FUNCTION_BLOCK FB_IdPool
VAR_INPUT
END_VAR
VAR_OUTPUT
END_VAR
VAR
	aNodes : ARRAY[1..cMaxObjects] OF ST_IdNode;
	pHead : POINTER TO ST_IdNode;
	pTail : POINTER TO ST_IdNode;
END_VAR

METHOD M_GetId : UINT
VAR_INPUT
END_VAR

VAR
	pNode : POINTER TO ST_IdNode;
END_VAR
IF pHead > 0 THEN
	pNode := pHead;
	M_GetId := pNode^.nId;
	IF pHead = pTail THEN //die letzte freie Id
		pHead := 0;
		pTail := 0;
	ELSE
		pHead := pNode^.pNext;
	END_IF
	memset(pNode,0,SIZEOF(ST_IdNode));
END_IF
END_METHOD

METHOD M_ReleaseId : BOOL
VAR_INPUT
	nId : UINT;
END_VAR
//Id in Benutzung?
IF nId >= 0 AND nId <= cMaxObjects AND_THEN aNodes[nId].nId = 0 THEN
	aNodes[nId].nId := nId;
	aNodes[nId].pNext := pHead;
	pHead := ADR(aNodes[nId]);
	M_ReleaseId := TRUE;
END_IF
END_METHOD

METHOD M_Reset : BOOL
VAR_INPUT
END_VAR

VAR
	i : UINT;
END_VAR
pHead := ADR(aNodes[1]);
pTail := ADR(aNodes[cMaxObjects]);
FOR i := 1 TO cMaxObjects BY 1 DO
	aNodes[i].nId := i;
	IF i < cMaxObjects THEN
		aNodes[i].pNext := ADR(aNodes[i+1]);
	ELSE
		aNodes[i].pNext := 0;
	END_IF
END_FOR
END_METHOD

END_FUNCTION_BLOCK

(* stored: Version 1.1.0.1, ProductVersion 3.1.4022.12
   POU FB_IdPool: Id {9849b2e5-dcee-4ced-81f0-c68734dbe188}, SpecialFunc None
   Method M_GetId: Id {e65a9dbd-6f70-4b71-8983-d548273ccf2e}
   Method M_ReleaseId: Id {99864b0b-dddb-4bbb-beb9-6636cb494557}
   Method M_Reset: Id {b1e69734-c5c2-4560-93fc-aafced5b842f} *)
